// TIA Portal V15.1 export
// export: Created 2024-05-17T05:38:38.0000355Z, ExportSetting WithDefaults, DisplayName Totally Integrated Automation Portal, DisplayVersion V15.1 Update 5, DisplayName TIA Portal Openness, DisplayVersion V15.1 Update 5, DisplayName SINAMICS Startdrive Advanced, DisplayVersion V15.1, DisplayName G130, G150, S120, S150, SINAMICS MV, S210, DisplayVersion V15.1, DisplayName G110M, G120, G120C, G120D, G120P, DisplayVersion V15.1, DisplayName STEP 7 Professional, DisplayVersion V15.1 Update 5, DisplayName STEP 7 Safety, DisplayVersion V15.1, DisplayName WinCC Professional, DisplayVersion V15.1 Update 5, DisplayName SIMATIC Visualization Architect, DisplayVersion V15.1
FUNCTION_BLOCK "LGBSEW-MoviProPN"   // FB6621, FBD
TITLE = LSEW-MoviProPN / LGBSEW-MoviProPN
{ S7_Optimized_Access := 'TRUE' }
VERSION : 0.1
// ============================================================================
// This module is the interface to a SEW drive MOVIPRO using universal telegram 10
// ============================================================================
// stored: AutoNumber false, IsIECCheckEnabled false, IsRetainMemResEnabled false, MemoryReserve 100, SetENOAutomatically False, UDAEnableTagReadback false
   VAR_INPUT
      I_ContolInhibit { ExternalAccessible := 'False'; ExternalVisible := 'False'; ExternalWritable := 'False'} : Bool;   // Inhibit motor (disable output stage, uncontolled stop)
      I_OFF1 { ExternalAccessible := 'False'; ExternalVisible := 'False'; ExternalWritable := 'False'} : Bool;   // start / stop motor
      I_OFF2 { ExternalAccessible := 'False'; ExternalVisible := 'False'; ExternalWritable := 'False'} : Bool := True;   // OFF2 rapid stop
      I_SetpointPosition { ExternalAccessible := 'False'; ExternalVisible := 'False'; ExternalWritable := 'False'} : DInt;   // Setpoint position [ user unit ex: rev. ]
      I_SetpointSpeed { ExternalAccessible := 'False'; ExternalVisible := 'False'; ExternalWritable := 'False'} : Int;   // Setpoint velocity [ user unit ex: rev./min ]
      I_Acceleration { ExternalAccessible := 'False'; ExternalVisible := 'False'; ExternalWritable := 'False'} : Int;   // Acceleration [ user unit ex: rev./(min*S) ]
      I_Deceleration { ExternalAccessible := 'False'; ExternalVisible := 'False'; ExternalWritable := 'False'} : Int;   // Deceleration [ user unit ex: rev./(min*S) ]
      I_ResetFault { ExternalAccessible := 'False'; ExternalVisible := 'False'; ExternalWritable := 'False'} : Bool;   // Reset fault
      I_BrakeRelease { ExternalAccessible := 'False'; ExternalVisible := 'False'; ExternalWritable := 'False'} : Bool;   // Command brake release
      I_OperatingMode { ExternalAccessible := 'False'; ExternalVisible := 'False'; ExternalWritable := 'False'} : USInt := 4;   // 0=Default, 1=Speed control, 2=Jog mode, 3=Referencing mode, 4=Positioning mode, 5=Positioning mode - touch probe, 6=Speed synchronization, 7=Emergency mode
      I_DisableSoftwareLimitSwitches { ExternalAccessible := 'False'; ExternalVisible := 'False'; ExternalWritable := 'False'} : Bool;   // Disable softwrare limit switches in the drive
      I_EnableTorqueLimiting { ExternalAccessible := 'False'; ExternalVisible := 'False'; ExternalWritable := 'False'} : Bool;   // Enable torque limiting
      I_JogPositive { ExternalAccessible := 'False'; ExternalVisible := 'False'; ExternalWritable := 'False'} : Bool;   // Jog in positive direction
      I_JogNegative { ExternalAccessible := 'False'; ExternalVisible := 'False'; ExternalWritable := 'False'} : Bool;   // Jog in negative direction
   END_VAR
   VAR_OUTPUT
      O_DriveReady { ExternalAccessible := 'False'; ExternalVisible := 'False'; ExternalWritable := 'False'} : Bool;   // Drive ready
      O_MaintenanceSwitch { ExternalAccessible := 'False'; ExternalVisible := 'False'; ExternalWritable := 'False'} : Bool;   // Maintenance switch activated (1=mains OFF)
      O_MotorTurning { ExternalAccessible := 'False'; ExternalVisible := 'False'; ExternalWritable := 'False'} : Bool;   // Motor turning
      O_SetpointReached { ExternalAccessible := 'False'; ExternalVisible := 'False'; ExternalWritable := 'False'} : Bool;   // Setpoint position is reached
      O_Referenced { ExternalAccessible := 'False'; ExternalVisible := 'False'; ExternalWritable := 'False'} : Bool;   // Drive is referenced
      O_HWLSPositive { ExternalAccessible := 'False'; ExternalVisible := 'False'; ExternalWritable := 'False'} : Bool;   // Hardware limit switch positive reached
      O_HWLSNegative { ExternalAccessible := 'False'; ExternalVisible := 'False'; ExternalWritable := 'False'} : Bool;   // Hardware limit switch negative reached
      O_Fault { ExternalAccessible := 'False'; ExternalVisible := 'False'; ExternalWritable := 'False'} : Bool;   // Fault present
      O_Warning { ExternalAccessible := 'False'; ExternalVisible := 'False'; ExternalWritable := 'False'} : Bool;   // Warning present
      O_ApplicationFault { ExternalAccessible := 'False'; ExternalVisible := 'False'; ExternalWritable := 'False'} : Bool;   // Application fault present
      O_Brake { ExternalAccessible := 'False'; ExternalVisible := 'False'; ExternalWritable := 'False'} : Bool;   // Brake status
      O_AliveBit { ExternalAccessible := 'False'; ExternalVisible := 'False'; ExternalWritable := 'False'} : Bool;   // Toggles default every 100ms
      H_StatusWord1 { ExternalAccessible := 'False'; ExternalVisible := 'False'; ExternalWritable := 'False'} : Word;   // Status word 1 from drive
      H_StatusWord2 { ExternalAccessible := 'False'; ExternalVisible := 'False'; ExternalWritable := 'False'} : Word;   // Status word 2 from drive
      H_StatusWord3 { ExternalAccessible := 'False'; ExternalVisible := 'False'; ExternalWritable := 'False'} : Word;   // Status word 3 from drive
      H_ControlWord1 { ExternalAccessible := 'False'; ExternalVisible := 'False'; ExternalWritable := 'False'} : Word;   // Control word 1 to drive
      H_ControlWord2 { ExternalAccessible := 'False'; ExternalVisible := 'False'; ExternalWritable := 'False'} : Word;   // Control word 2 to drive
      H_SetpointPosition { ExternalAccessible := 'False'; ExternalVisible := 'False'; ExternalWritable := 'False'} : DInt;   // Setpoint position [ user unit ex: rev. ]
      H_SetpointSpeed { ExternalAccessible := 'False'; ExternalVisible := 'False'; ExternalWritable := 'False'} : Int;   // Setpoint velocity [ user unit ex: rev./min ]
      H_Acceleration { ExternalAccessible := 'False'; ExternalVisible := 'False'; ExternalWritable := 'False'} : Int;   // Acceleration [ user unit ex: rev./(min*S) ]
      H_Deceleration { ExternalAccessible := 'False'; ExternalVisible := 'False'; ExternalWritable := 'False'} : Int;   // Deceleration [ user unit ex: rev./(min*S) ]
      H_ActualSpeed { ExternalAccessible := 'False'; ExternalVisible := 'False'; ExternalWritable := 'False'} : Int;   // Actual velocity [ user unit ex: rev./min ]
      H_ActualPosition { ExternalAccessible := 'False'; ExternalVisible := 'False'; ExternalWritable := 'False'} : DInt;   // Actual position [ user unit ex: rev. ]
      H_ActualCurrentA { ExternalAccessible := 'False'; ExternalVisible := 'False'; ExternalWritable := 'False'} : Real;   // Actual current Ampere
      "H_ActualCurrent%" { ExternalAccessible := 'False'; ExternalVisible := 'False'; ExternalWritable := 'False'} : Real;   // Actual current %
      H_ActualWarning { ExternalAccessible := 'False'; ExternalVisible := 'False'; ExternalWritable := 'False'} : Int;   // Actual Warning From Drive
      H_ActualFault { ExternalAccessible := 'False'; ExternalVisible := 'False'; ExternalWritable := 'False'} : Int;   // Actual Fault From Drive
   END_VAR
   VAR_IN_OUT
      C_HWSubInput { ExternalAccessible := 'False'; ExternalVisible := 'False'; ExternalWritable := 'False'} : HW_SUBMODULE;   // Inputs telegram 10 Hardware identifier
      C_HWSubOutput { ExternalAccessible := 'False'; ExternalVisible := 'False'; ExternalWritable := 'False'} : HW_SUBMODULE;   // Outputs telegram 10 Hardware identifier
      C_HWSubControllerInput { ExternalAccessible := 'False'; ExternalVisible := 'False'; ExternalWritable := 'False'} : HW_SUBMODULE;   // Controller inputs telegram 2 Hardware identifier
      C_HWSubControllerOutput { ExternalAccessible := 'False'; ExternalVisible := 'False'; ExternalWritable := 'False'} : HW_SUBMODULE;   // Controller outputs telegram 2 Hardware identifier
      C_DriveCurrent { ExternalAccessible := 'False'; ExternalVisible := 'False'; ExternalWritable := 'False'} : Real;   // Reference current of the drive
      C_MotorCurrent { ExternalAccessible := 'False'; ExternalVisible := 'False'; ExternalWritable := 'False'} : Real;   // Reference current of the motor
   END_VAR
   VAR
      InputTelegram { ExternalAccessible := 'False'; ExternalVisible := 'False'; ExternalWritable := 'False'} : "SEW_MOVIPRO_Universal_TEL_10_Inputs";   // Input telegram
      OutputTelegram { ExternalAccessible := 'False'; ExternalVisible := 'False'; ExternalWritable := 'False'} : "SEW_MOVIPRO_Universal_TEL_10_Outputs";   // Output telegram
      ControllerInputTelegram { ExternalAccessible := 'False'; ExternalVisible := 'False'; ExternalWritable := 'False'} : "SEW_MOVIPRO_Controller_TEL_2_Inputs";   // Controller input telegram
      ControllerOutputTelegram { ExternalAccessible := 'False'; ExternalVisible := 'False'; ExternalWritable := 'False'} : "SEW_MOVIPRO_Controller_TEL_2_Outputs";   // Controller output telegram
      OperatingMode { ExternalAccessible := 'False'; ExternalVisible := 'False'; ExternalWritable := 'False'} : USInt;   // Operating mode
   END_VAR
   VAR_TEMP
      TempReal : Real;   // Temp Real
      "Comment#1" : Bool;
   END_VAR
BEGIN

REGION Network 1: **** 1 - Inputs **** Read input telegram and store in struct
   // Copies the Input telegram to a local varibale struct
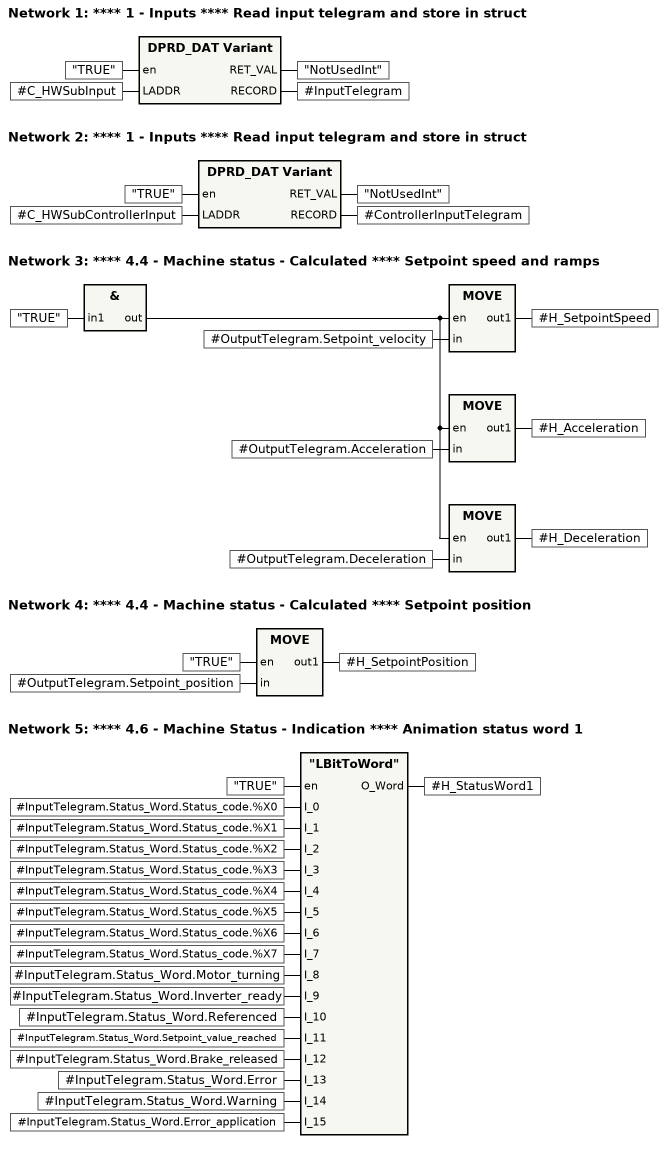
   IF "TRUE" THEN
       "NotUsedInt" := DPRD_DAT(LADDR := #C_HWSubInput, RECORD => #InputTelegram);   // Copy data with HW ID SEW Drive ______________ ll __ _ ll__ input telegram ll l__l l_l ll Ol ===============>> PLC ll ll__l ll_____________ll l__l l__l l_ll_l _
   END_IF;
END_REGION

REGION Network 2: **** 1 - Inputs **** Read input telegram and store in struct
   // Copies the Input telegram to a local varibale struct
   IF "TRUE" THEN
       "NotUsedInt" := DPRD_DAT(LADDR := #C_HWSubControllerInput, RECORD => #ControllerInputTelegram);   // Copy data with HW ID SEW Drive ______________ ll __ _ ll__ input telegram ll l__l l_l ll Ol ===============>> PLC ll ll__l ll_____________ll l__l l__l l_ll_l _
   END_IF;
END_REGION

REGION Network 3: **** 4.4 - Machine status - Calculated **** Setpoint speed and ramps
   // Convert Data
   IF "TRUE" THEN
       #H_SetpointSpeed := #OutputTelegram.Setpoint_velocity;
       #H_Acceleration := #OutputTelegram.Acceleration;
       #H_Deceleration := #OutputTelegram.Deceleration;
   END_IF;
END_REGION

REGION Network 4: **** 4.4 - Machine status - Calculated **** Setpoint position
   // Convert Data
   IF "TRUE" THEN #H_SetpointPosition := #OutputTelegram.Setpoint_position; END_IF;
END_REGION

REGION Network 5: **** 4.6 - Machine Status - Indication **** Animation status word 1
   // Animation
   IF "TRUE" THEN
       "LBitToWord"(I_0 := #InputTelegram.Status_Word.Status_code.%X0,   // HMI PLC __________________________________________________________ l _SIEMENS____________________________SIMATIC HMI_____ l ___________________ l l l l l_l_l_l______________l l l l l l SIEMENS SIMATIC l l l ________________ l l l ________S7-1500 l l l l_____________ X l l l l l___________O_l l l l l l l l l l l l l l l Popup or l l l l l l l l l l screen. l l l l l l l l l l l <<-------==================l= l========= l l l l l l l Anim l l l l l______________l l l l l_______________l l l l ___ l l l l l l __l l__ l l l l l l l__ __l l l l l l l l___l l l l l l l l l l_____________________________________________________ l l l__________________ l l_________________________________________________________ l Animation word is send to the HMI to be used in object screen or popup _
                    I_1 := #InputTelegram.Status_Word.Status_code.%X1,
                    I_2 := #InputTelegram.Status_Word.Status_code.%X2,
                    I_3 := #InputTelegram.Status_Word.Status_code.%X3,
                    I_4 := #InputTelegram.Status_Word.Status_code.%X4,
                    I_5 := #InputTelegram.Status_Word.Status_code.%X5,
                    I_6 := #InputTelegram.Status_Word.Status_code.%X6,
                    I_7 := #InputTelegram.Status_Word.Status_code.%X7,
                    I_8 := #InputTelegram.Status_Word.Motor_turning,
                    I_9 := #InputTelegram.Status_Word.Inverter_ready,
                    I_10 := #InputTelegram.Status_Word.Referenced,
                    I_11 := #InputTelegram.Status_Word.Setpoint_value_reached,
                    I_12 := #InputTelegram.Status_Word.Brake_released,
                    I_13 := #InputTelegram.Status_Word.Error,
                    I_14 := #InputTelegram.Status_Word.Warning,
                    I_15 := #InputTelegram.Status_Word.Error_application,
                    O_Word => #H_StatusWord1);
   END_IF;
END_REGION

REGION Network 6: **** 4.6 - Machine Status - Indication **** Animation status word 2
   // Animation
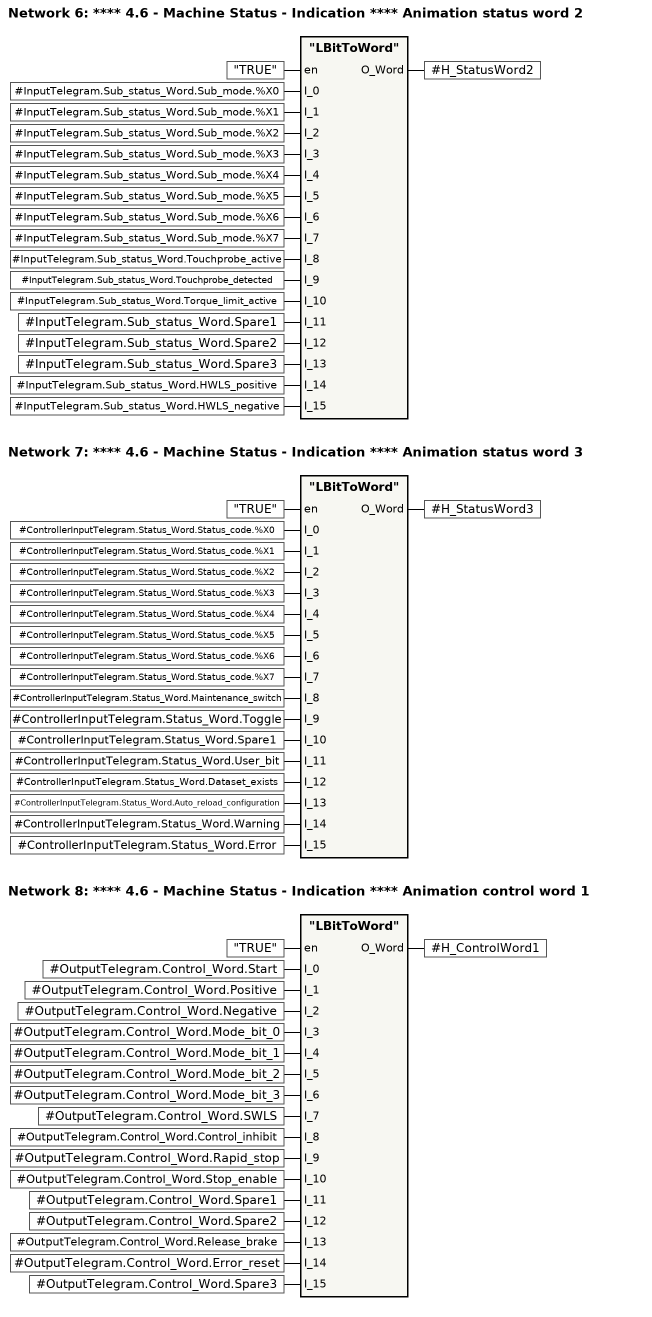
   IF "TRUE" THEN
       "LBitToWord"(I_0 := #InputTelegram.Sub_status_Word.Sub_mode.%X0,   // HMI PLC __________________________________________________________ l _SIEMENS____________________________SIMATIC HMI_____ l ___________________ l l l l l_l_l_l______________l l l l l l SIEMENS SIMATIC l l l ________________ l l l ________S7-1500 l l l l_____________ X l l l l l___________O_l l l l l l l l l l l l l l l Popup or l l l l l l l l l l screen. l l l l l l l l l l l <<-------==================l= l========= l l l l l l l Anim l l l l l______________l l l l l_______________l l l l ___ l l l l l l __l l__ l l l l l l l__ __l l l l l l l l___l l l l l l l l l l_____________________________________________________ l l l__________________ l l_________________________________________________________ l Animation word is send to the HMI to be used in object screen or popup _
                    I_1 := #InputTelegram.Sub_status_Word.Sub_mode.%X1,
                    I_2 := #InputTelegram.Sub_status_Word.Sub_mode.%X2,
                    I_3 := #InputTelegram.Sub_status_Word.Sub_mode.%X3,
                    I_4 := #InputTelegram.Sub_status_Word.Sub_mode.%X4,
                    I_5 := #InputTelegram.Sub_status_Word.Sub_mode.%X5,
                    I_6 := #InputTelegram.Sub_status_Word.Sub_mode.%X6,
                    I_7 := #InputTelegram.Sub_status_Word.Sub_mode.%X7,
                    I_8 := #InputTelegram.Sub_status_Word.Touchprobe_active,
                    I_9 := #InputTelegram.Sub_status_Word.Touchprobe_detected,
                    I_10 := #InputTelegram.Sub_status_Word.Torque_limit_active,
                    I_11 := #InputTelegram.Sub_status_Word.Spare1,
                    I_12 := #InputTelegram.Sub_status_Word.Spare2,
                    I_13 := #InputTelegram.Sub_status_Word.Spare3,
                    I_14 := #InputTelegram.Sub_status_Word.HWLS_positive,
                    I_15 := #InputTelegram.Sub_status_Word.HWLS_negative,
                    O_Word => #H_StatusWord2);
   END_IF;
END_REGION

REGION Network 7: **** 4.6 - Machine Status - Indication **** Animation status word 3
   // Animation
   IF "TRUE" THEN
       "LBitToWord"(I_0 := #ControllerInputTelegram.Status_Word.Status_code.%X0,   // HMI PLC __________________________________________________________ l _SIEMENS____________________________SIMATIC HMI_____ l ___________________ l l l l l_l_l_l______________l l l l l l SIEMENS SIMATIC l l l ________________ l l l ________S7-1500 l l l l_____________ X l l l l l___________O_l l l l l l l l l l l l l l l Popup or l l l l l l l l l l screen. l l l l l l l l l l l <<-------==================l= l========= l l l l l l l Anim l l l l l______________l l l l l_______________l l l l ___ l l l l l l __l l__ l l l l l l l__ __l l l l l l l l___l l l l l l l l l l_____________________________________________________ l l l__________________ l l_________________________________________________________ l Animation word is send to the HMI to be used in object screen or popup _
                    I_1 := #ControllerInputTelegram.Status_Word.Status_code.%X1,
                    I_2 := #ControllerInputTelegram.Status_Word.Status_code.%X2,
                    I_3 := #ControllerInputTelegram.Status_Word.Status_code.%X3,
                    I_4 := #ControllerInputTelegram.Status_Word.Status_code.%X4,
                    I_5 := #ControllerInputTelegram.Status_Word.Status_code.%X5,
                    I_6 := #ControllerInputTelegram.Status_Word.Status_code.%X6,
                    I_7 := #ControllerInputTelegram.Status_Word.Status_code.%X7,
                    I_8 := #ControllerInputTelegram.Status_Word.Maintenance_switch,
                    I_9 := #ControllerInputTelegram.Status_Word.Toggle,
                    I_10 := #ControllerInputTelegram.Status_Word.Spare1,
                    I_11 := #ControllerInputTelegram.Status_Word.User_bit,
                    I_12 := #ControllerInputTelegram.Status_Word.Dataset_exists,
                    I_13 := #ControllerInputTelegram.Status_Word.Auto_reload_configuration,
                    I_14 := #ControllerInputTelegram.Status_Word.Warning,
                    I_15 := #ControllerInputTelegram.Status_Word.Error,
                    O_Word => #H_StatusWord3);
   END_IF;
END_REGION

REGION Network 8: **** 4.6 - Machine Status - Indication **** Animation control word 1
   // Animation
   IF "TRUE" THEN
       "LBitToWord"(I_0 := #OutputTelegram.Control_Word.Start,   // HMI PLC __________________________________________________________ l _SIEMENS____________________________SIMATIC HMI_____ l ___________________ l l l l l_l_l_l______________l l l l l l SIEMENS SIMATIC l l l ________________ l l l ________S7-1500 l l l l_____________ X l l l l l___________O_l l l l l l l l l l l l l l l Popup or l l l l l l l l l l screen. l l l l l l l l l l l <<-------==================l= l========= l l l l l l l Anim l l l l l______________l l l l l_______________l l l l ___ l l l l l l __l l__ l l l l l l l__ __l l l l l l l l___l l l l l l l l l l_____________________________________________________ l l l__________________ l l_________________________________________________________ l Animation word is send to the HMI to be used in object screen or popup _
                    I_1 := #OutputTelegram.Control_Word.Positive,
                    I_2 := #OutputTelegram.Control_Word.Negative,
                    I_3 := #OutputTelegram.Control_Word.Mode_bit_0,
                    I_4 := #OutputTelegram.Control_Word.Mode_bit_1,
                    I_5 := #OutputTelegram.Control_Word.Mode_bit_2,
                    I_6 := #OutputTelegram.Control_Word.Mode_bit_3,
                    I_7 := #OutputTelegram.Control_Word.SWLS,
                    I_8 := #OutputTelegram.Control_Word.Control_inhibit,
                    I_9 := #OutputTelegram.Control_Word.Rapid_stop,
                    I_10 := #OutputTelegram.Control_Word.Stop_enable,
                    I_11 := #OutputTelegram.Control_Word.Spare1,
                    I_12 := #OutputTelegram.Control_Word.Spare2,
                    I_13 := #OutputTelegram.Control_Word.Release_brake,
                    I_14 := #OutputTelegram.Control_Word.Error_reset,
                    I_15 := #OutputTelegram.Control_Word.Spare3,
                    O_Word => #H_ControlWord1);
   END_IF;
END_REGION

REGION Network 9: **** 4.6 - Machine Status - Indication **** Animation control word 2
   // Animation
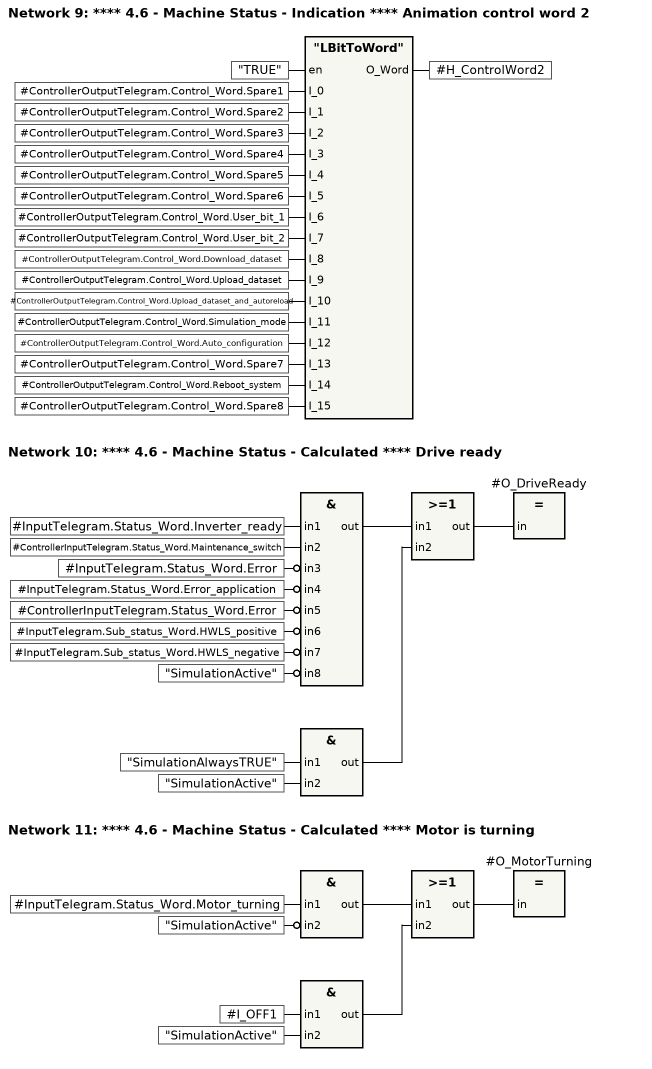
   IF "TRUE" THEN
       "LBitToWord"(I_0 := #ControllerOutputTelegram.Control_Word.Spare1,   // HMI PLC __________________________________________________________ l _SIEMENS____________________________SIMATIC HMI_____ l ___________________ l l l l l_l_l_l______________l l l l l l SIEMENS SIMATIC l l l ________________ l l l ________S7-1500 l l l l_____________ X l l l l l___________O_l l l l l l l l l l l l l l l Popup or l l l l l l l l l l screen. l l l l l l l l l l l <<-------==================l= l========= l l l l l l l Anim l l l l l______________l l l l l_______________l l l l ___ l l l l l l __l l__ l l l l l l l__ __l l l l l l l l___l l l l l l l l l l_____________________________________________________ l l l__________________ l l_________________________________________________________ l Animation word is send to the HMI to be used in object screen or popup _
                    I_1 := #ControllerOutputTelegram.Control_Word.Spare2,
                    I_2 := #ControllerOutputTelegram.Control_Word.Spare3,
                    I_3 := #ControllerOutputTelegram.Control_Word.Spare4,
                    I_4 := #ControllerOutputTelegram.Control_Word.Spare5,
                    I_5 := #ControllerOutputTelegram.Control_Word.Spare6,
                    I_6 := #ControllerOutputTelegram.Control_Word.User_bit_1,
                    I_7 := #ControllerOutputTelegram.Control_Word.User_bit_2,
                    I_8 := #ControllerOutputTelegram.Control_Word.Download_dataset,
                    I_9 := #ControllerOutputTelegram.Control_Word.Upload_dataset,
                    I_10 := #ControllerOutputTelegram.Control_Word.Upload_dataset_and_autoreload,
                    I_11 := #ControllerOutputTelegram.Control_Word.Simulation_mode,
                    I_12 := #ControllerOutputTelegram.Control_Word.Auto_configuration,
                    I_13 := #ControllerOutputTelegram.Control_Word.Spare7,
                    I_14 := #ControllerOutputTelegram.Control_Word.Reboot_system,
                    I_15 := #ControllerOutputTelegram.Control_Word.Spare8,
                    O_Word => #H_ControlWord2);
   END_IF;
END_REGION

REGION Network 10: **** 4.6 - Machine Status - Calculated **** Drive ready
   // Drive ready state and no alarms are active
   #O_DriveReady := (#InputTelegram.Status_Word.Inverter_ready AND #ControllerInputTelegram.Status_Word.Maintenance_switch AND NOT #InputTelegram.Status_Word.Error AND NOT #InputTelegram.Status_Word.Error_application AND NOT #ControllerInputTelegram.Status_Word.Error AND NOT #InputTelegram.Sub_status_Word.HWLS_positive AND NOT #InputTelegram.Sub_status_Word.HWLS_negative AND NOT "SimulationActive") OR ("SimulationAlwaysTRUE" AND "SimulationActive");
END_REGION

REGION Network 11: **** 4.6 - Machine Status - Calculated **** Motor is turning
   // Ouput stage enabled (motor powered)
   #O_MotorTurning := (#InputTelegram.Status_Word.Motor_turning AND NOT "SimulationActive") OR (#I_OFF1 AND "SimulationActive");
END_REGION

REGION Network 12: **** 4.6 - Machine Status - Calculated **** Status / Warning / Fault code from drive
   // When the fault input is "True"   then the status code send over the byte is a fault code as decimal.
   // When the fault input is "False" then the status code send over the byte is a warning / status code as decimal.
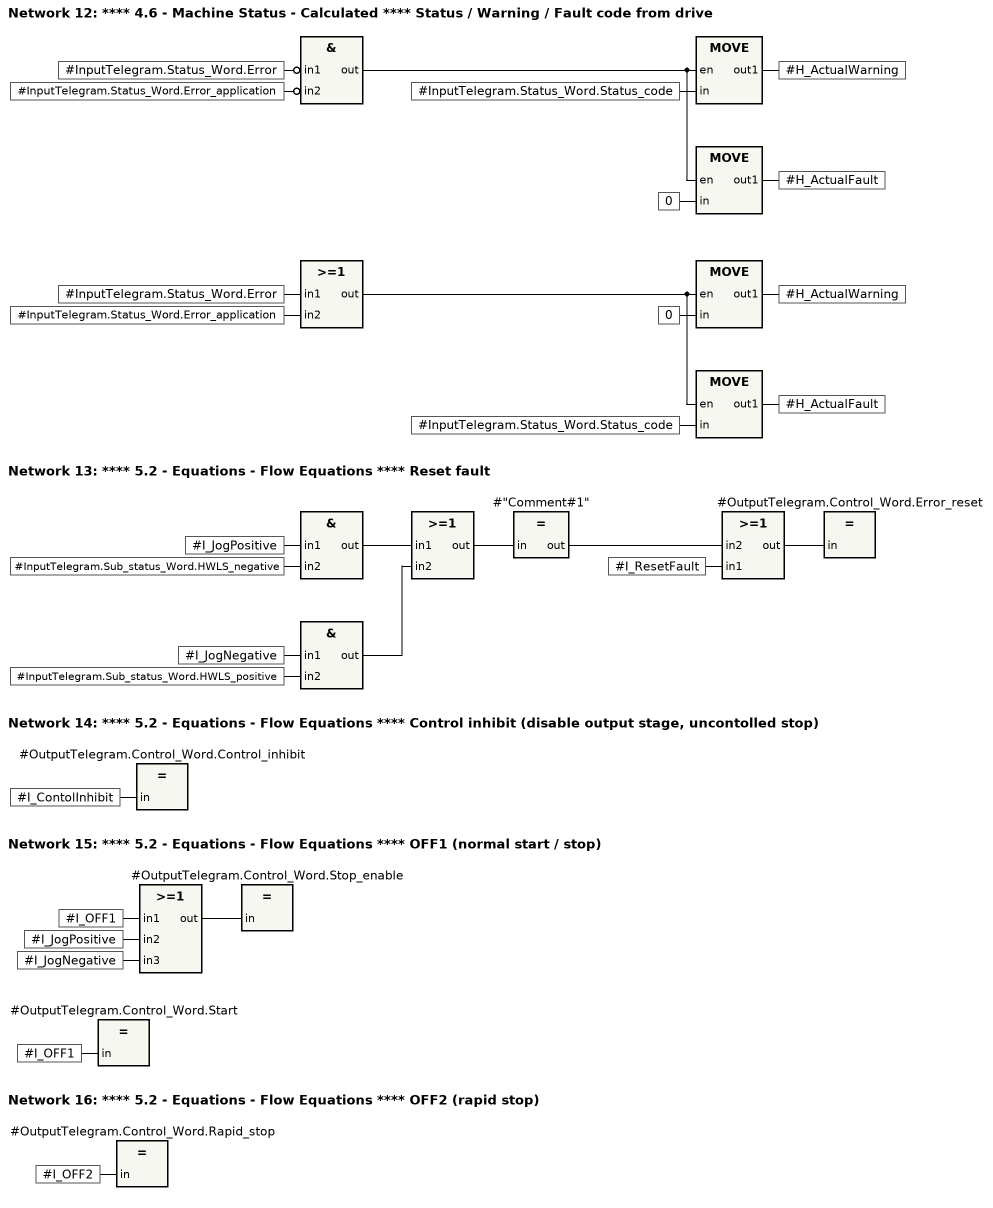
   IF NOT #InputTelegram.Status_Word.Error AND NOT #InputTelegram.Status_Word.Error_application THEN
       #H_ActualWarning := #InputTelegram.Status_Word.Status_code;
       #H_ActualFault := 0;
   END_IF;
   IF #InputTelegram.Status_Word.Error OR #InputTelegram.Status_Word.Error_application THEN
       #H_ActualWarning := 0;
       #H_ActualFault := #InputTelegram.Status_Word.Status_code;
   END_IF;
END_REGION

REGION Network 13: **** 5.2 - Equations - Flow Equations **** Reset fault
   #"Comment#1" := (#I_JogPositive AND #InputTelegram.Sub_status_Word.HWLS_negative) OR (#I_JogNegative AND #InputTelegram.Sub_status_Word.HWLS_positive);   // Reset fault will cause the motor to turn out of the currently active limitswitch. This is coupled with the JOG Function in the direction away from the limit switch.
   #OutputTelegram.Control_Word.Error_reset := #"Comment#1" OR #I_ResetFault;
END_REGION

REGION Network 14: **** 5.2 - Equations - Flow Equations **** Control inhibit (disable output stage, uncontolled stop)
   #OutputTelegram.Control_Word.Control_inhibit := #I_ContolInhibit;
END_REGION

REGION Network 15: **** 5.2 - Equations - Flow Equations **** OFF1 (normal start / stop)
   #OutputTelegram.Control_Word.Stop_enable := #I_OFF1 OR #I_JogPositive OR #I_JogNegative;
   #OutputTelegram.Control_Word.Start := #I_OFF1;
END_REGION

REGION Network 16: **** 5.2 - Equations - Flow Equations **** OFF2 (rapid stop)
   #OutputTelegram.Control_Word.Rapid_stop := #I_OFF2;   // ^ Speed (%) Stop signal at 5s l / 100% l______________/_ l \ \ l \ \ l \ \ l \ \ 0% l___________________\_____\___________________________> Time (s) l OFF2 OFF1 (regular start stop) 7s 10s Ramp down time settings to be done in the drive. OFF2 is to be used for controlled stops when there is a need to stop faster then regular, for example when there is an E-stop at a lift it is better to do a controlled stop and after that (x time in safety program) to give a STO. Note if there is a safe stop availible on safety level this is to be used instead of the non safety signals. _
END_REGION

REGION Network 17: **** 5.2 - Equations - Flow Equations **** Setpoint Speed and ramps
   // Setpoint speed in user unit's (ex. 100mm/s)
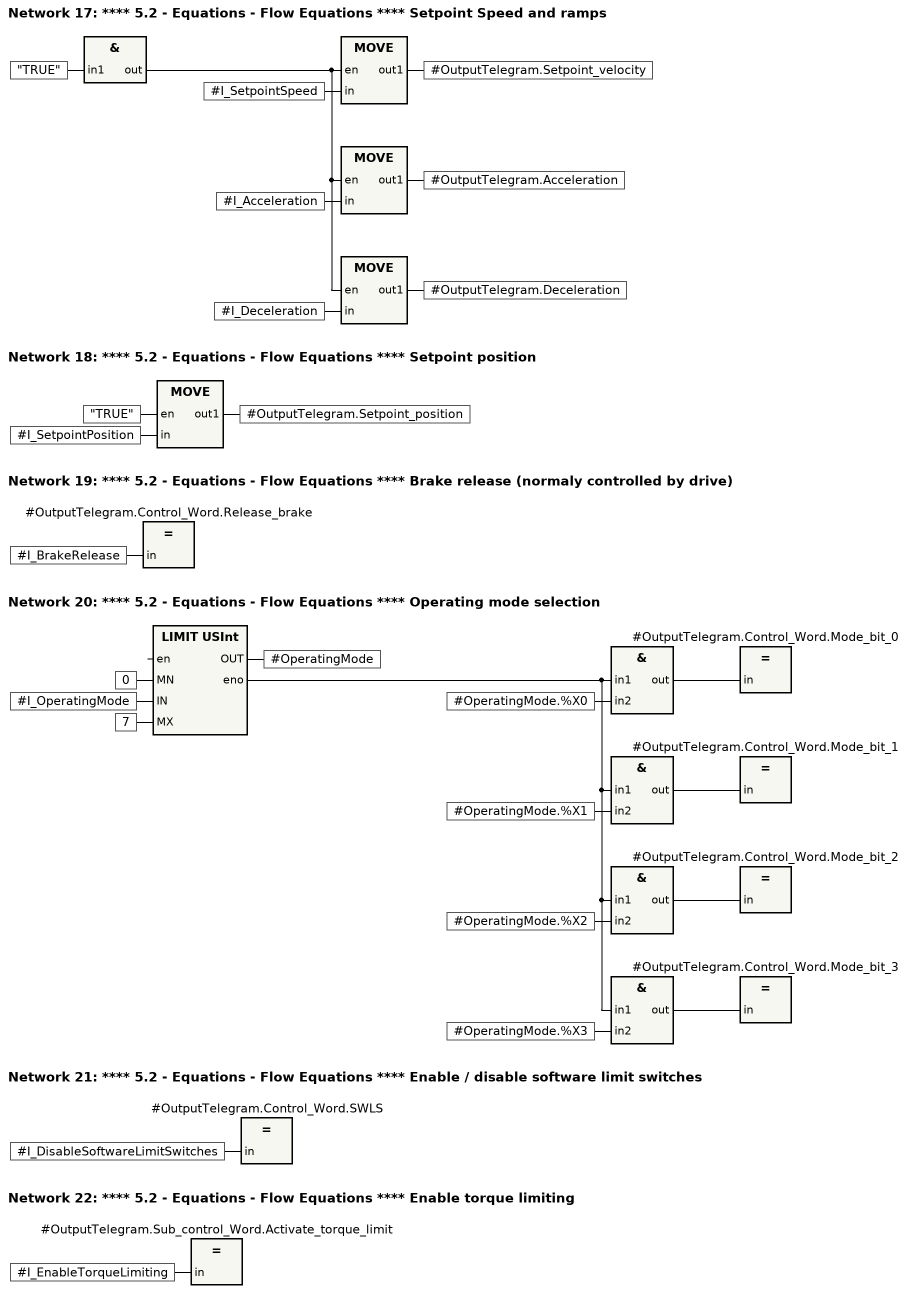
   IF "TRUE" THEN
       #OutputTelegram.Setpoint_velocity := #I_SetpointSpeed;   // Speed Target speed (user unit) ^ / l ____/____ l / \ l / \ l____/ \____ l--------------------------------------------------> t (s) _
       #OutputTelegram.Acceleration := #I_Acceleration;   // Speed (user unit) ^ Acceleration l l _________ l l / \ l l/ \ l____/ \____ l--------------------------------------------------> t (s) _
       #OutputTelegram.Deceleration := #I_Deceleration;   // Speed (user unit) ^ Deceleration l _________ l l / \ l l / \l l____/ \____ l--------------------------------------------------> t (s) _
   END_IF;
END_REGION

REGION Network 18: **** 5.2 - Equations - Flow Equations **** Setpoint position
   // Setpoint position [ user unit ex: rev. ] (ex. 13490mm)
   IF "TRUE" THEN
       #OutputTelegram.Setpoint_position := #I_SetpointPosition;   // Setpoint position [ user unit ex: rev. ] (ex. 13490mm) / / / / /_/______/_/ _________ /_/_____/_/ l /_/_____/_/ l --> Level +13,49 /_/_____/_/ l l l l l l l l l l l l l l l l l l l l l l l l l l l l l l l l l l l l l l l l l l l l l l l l l l l l l l l l l l l l l l l______l_ l l /_/_____/l_/ --> Level +7,06 l/_/_____/ l/ l_/_____/_l _________ / / / / / / / /
   END_IF;
END_REGION

REGION Network 19: **** 5.2 - Equations - Flow Equations **** Brake release (normaly controlled by drive)
   // Brake release (normaly controlled by drive), Possibility to release brake at any moment.
   #OutputTelegram.Control_Word.Release_brake := #I_BrakeRelease;   // Not to be used for normal operation!!! In normal operation this is done by the drive.
END_REGION

REGION Network 20: **** 5.2 - Equations - Flow Equations **** Operating mode selection
   #OperatingMode := LIMIT(MN := 0, IN := #I_OperatingMode, MX := 7);   // Limit mode selection between 0 and 7. Then copy the booleans to the output telegram for the drive. "OperatingMode" --> Output telegram (Byte) (mode booleans) 0 ------> 0 0 ------> 0 0 ------> 0 0 ------> 0 0 0 0 0
   #OutputTelegram.Control_Word.Mode_bit_0 := #OperatingMode.%X0;   // Mode selection bits mode: 0=Default 1=Speed control 2=Jog mode 3=Referencing mode 4=Positioning mode 5=Positioning mode - touch probe 6=Speed synchronization 7=Emergency mode
   #OutputTelegram.Control_Word.Mode_bit_1 := #OperatingMode.%X1;
   #OutputTelegram.Control_Word.Mode_bit_2 := #OperatingMode.%X2;
   #OutputTelegram.Control_Word.Mode_bit_3 := #OperatingMode.%X3;
END_REGION

REGION Network 21: **** 5.2 - Equations - Flow Equations **** Enable / disable software limit switches
   #OutputTelegram.Control_Word.SWLS := #I_DisableSoftwareLimitSwitches;   // Software limit switches: The software limit switches are programmed before the hardware limit switches. This will give the drive the possiblility to decelarate accordingly as its knows the distance to these SW LS's from the encoder value. When the referencing is ok it should be impossible to reach the hardware limit switches. Only when there is a faulty referencing then the software limit switches can be behind the hardware limit switch. In that case it is possible to hit the hardware limit switch with full speed. Positive <-- Load --> negative HW LS SW LS _____ SW LS HW LS ____ ____ l_____l ____ ____ l____\ l____\ l_____l /____l /____l OOOOOOOOOOOOOOOOOOOOOOOOOOOOOOOOOOOO ll // \\ ll ll// \\ll ll ll _
END_REGION

REGION Network 22: **** 5.2 - Equations - Flow Equations **** Enable torque limiting
   #OutputTelegram.Sub_control_Word.Activate_torque_limit := #I_EnableTorqueLimiting;   // 110% ^ Torque (%) l Torque limited 100% l_______________________________/___________________ torque limit configured in the drive l _ Acceleration l l l l l / l l---- shutdown command l l l/ constant speed l l (error motor blocked) l l l_____/__ l l 0% l___l_________l________________l__l___________________________> Time (s) l l l l l l l / l l l / l_l -100% l __________ /________________________________________ torque limit configured in the drive l Deceleration -110% l _
END_REGION

REGION Network 23 (SCL): **** 5.2 - Equations - Flow Equations **** Not used booleans (always FALSE)
   // Output variables that are not used are written constantly to False or 0.

   #OutputTelegram.Sub_control_Word.Activate_touchprobe := False;
   #ControllerOutputTelegram.Control_Word.User_bit_1 := False;
   #ControllerOutputTelegram.Control_Word.User_bit_2 := False;
   #ControllerOutputTelegram.Control_Word.Download_dataset := False;
   #ControllerOutputTelegram.Control_Word.Upload_dataset := False;
   #ControllerOutputTelegram.Control_Word.Upload_dataset_and_autoreload := False;
   #ControllerOutputTelegram.Control_Word.Simulation_mode := False;
   #ControllerOutputTelegram.Control_Word.Auto_configuration := False;
   #ControllerOutputTelegram.Control_Word.Reboot_system := False;
END_REGION

REGION Network 24: **** 8 - Outputs ****Motor Current
   // Motor Current in % compared to the drive reference current (not the motor reference current)
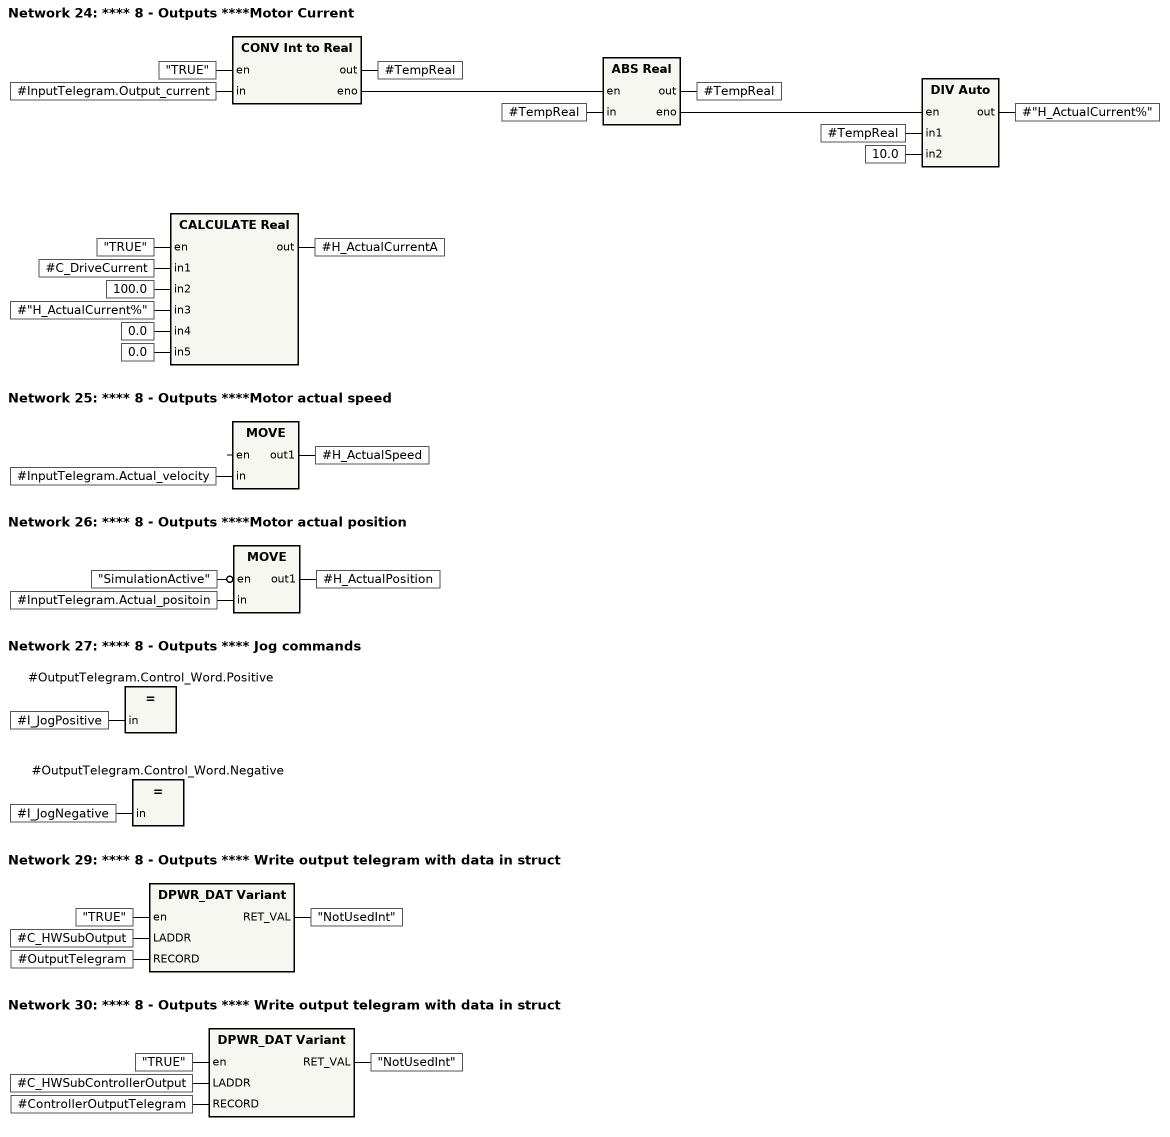
   IF "TRUE" THEN
       #TempReal := INT_TO_REAL(#InputTelegram.Output_current);
       #TempReal := ABS(#TempReal);   // Motor Current in % compared to the drive reference current (not the motor reference current) Remove - sign and use absolute value. Then scale this to the correct value (divide by 10 to get %) (This needs to be done since the drive can only send intiger values and not real values, so the drive does the percentage x10 to give a value behind the comma.) Then scale the % to a Ampere value and a % value compared to the motor reference current.
       #"H_ActualCurrent%" := #TempReal / 10.0;
       #H_ActualCurrentA := #C_DriveCurrent - (((100.0 - #"H_ActualCurrent%") / (100.0 - 0.0)) * (#C_DriveCurrent- 0.0));
   END_IF;
END_REGION

REGION Network 25: **** 8 - Outputs ****Motor actual speed
   #H_ActualSpeed := #InputTelegram.Actual_velocity;
END_REGION

REGION Network 26: **** 8 - Outputs ****Motor actual position
   IF NOT "SimulationActive" THEN #H_ActualPosition := #InputTelegram.Actual_positoin; END_IF;
END_REGION

REGION Network 27: **** 8 - Outputs **** Jog commands
   #OutputTelegram.Control_Word.Positive := #I_JogPositive;
   #OutputTelegram.Control_Word.Negative := #I_JogNegative;
END_REGION

REGION Network 28 (SCL): **** 8 - Outputs **** Status / Fault booleans
   // Copy input telegram booleans to O_****** parameters for use outside this block.

   #O_MaintenanceSwitch := #ControllerInputTelegram.Status_Word.Maintenance_switch;
   #O_AliveBit := #ControllerInputTelegram.Status_Word.Toggle;
   #O_Referenced := #InputTelegram.Status_Word.Referenced;
   IF NOT "SimulationActive" THEN
       #O_SetpointReached := #InputTelegram.Status_Word.Setpoint_value_reached;
   ELSE
       #O_SetpointReached := "SimulationAlwaysTRUE";
   END_IF;
   #O_Brake := #InputTelegram.Status_Word.Brake_released;
   #O_Fault := #InputTelegram.Status_Word.Error OR #ControllerInputTelegram.Status_Word.Error;
   #O_Warning := #InputTelegram.Status_Word.Warning OR #ControllerInputTelegram.Status_Word.Warning;
   #O_ApplicationFault := #InputTelegram.Status_Word.Error_application;
   #O_HWLSPositive := #InputTelegram.Sub_status_Word.HWLS_positive;
   #O_HWLSNegative := #InputTelegram.Sub_status_Word.HWLS_negative;
END_REGION

REGION Network 29: **** 8 - Outputs **** Write output telegram with data in struct
   IF "TRUE" THEN
       "NotUsedInt" := DPWR_DAT(LADDR := #C_HWSubOutput, RECORD := #OutputTelegram);   // Copy data with HW ID SEW Drive ______________ output telegram ll __ _ ll__ PLC ===============>> ll l__l l_l ll Ol ll ll__l ll_____________ll l__l l__l l_ll_l _
   END_IF;
END_REGION

REGION Network 30: **** 8 - Outputs **** Write output telegram with data in struct
   IF "TRUE" THEN
       "NotUsedInt" := DPWR_DAT(LADDR := #C_HWSubControllerOutput, RECORD := #ControllerOutputTelegram);   // Copy data with HW ID SEW Drive ______________ output telegram ll __ _ ll__ PLC ===============>> ll l__l l_l ll Ol ll ll__l ll_____________ll l__l l__l l_ll_l _
   END_IF;
END_REGION
END_FUNCTION_BLOCK
